PROGRAM Axis02_Status
VAR
//System_Bit
	Always_ON	:	BOOL	:=TRUE	;//상시 ON 
	Always_OFF	:	BOOL	:=FALSE	;//상시 OFF
	
//Motor_Command
	Axis02_Status_01: MC_ReadStatus;
	Axis02_Position_Read_01: MC_ReadActualPosition;
	Axis02_Velocity_Read_01: MC_ReadActualVelocity;
	Axis02_Reset_01: MC_Reset;
	Axis02_Stop_01: MC_Stop;
END_VAR

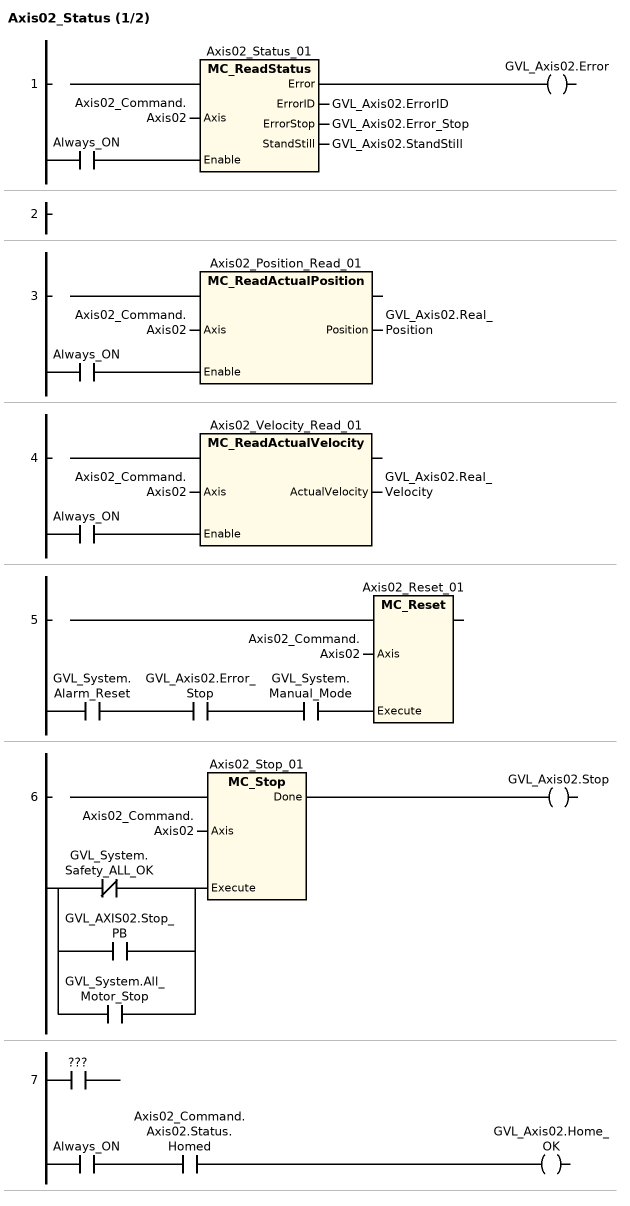
// NETWORK 1
Axis02_Status_01(
    Axis := Axis02_Command.Axis02,
    Enable := Always_ON,
    Error => GVL_Axis02.Error,
    ErrorID => GVL_Axis02.ErrorID,
    ErrorStop => GVL_Axis02.Error_Stop,
    StandStill => GVL_Axis02.StandStill); // MC_ReadStatus

// NETWORK 2

// NETWORK 3
Axis02_Position_Read_01(
    Axis := Axis02_Command.Axis02,
    Enable := Always_ON,
    Position => GVL_Axis02.Real_Position); // MC_ReadActualPosition

// NETWORK 4
Axis02_Velocity_Read_01(
    Axis := Axis02_Command.Axis02,
    Enable := Always_ON,
    ActualVelocity => GVL_Axis02.Real_Velocity); // MC_ReadActualVelocity

// NETWORK 5
Axis02_Reset_01(Axis := Axis02_Command.Axis02, Execute := GVL_System.Alarm_Reset AND GVL_Axis02.Error_Stop AND GVL_System.Manual_Mode); // MC_Reset

// NETWORK 6
Axis02_Stop_01(Axis := Axis02_Command.Axis02, Execute := NOT GVL_System.Safety_ALL_OK OR GVL_AXIS02.Stop_PB OR GVL_System.All_Motor_Stop); // MC_Stop
GVL_Axis02.Stop := Axis02_Stop_01.Done;

// NETWORK 7
GVL_Axis02.Home_OK := Always_ON AND Axis02_Command.Axis02.Status.Homed;

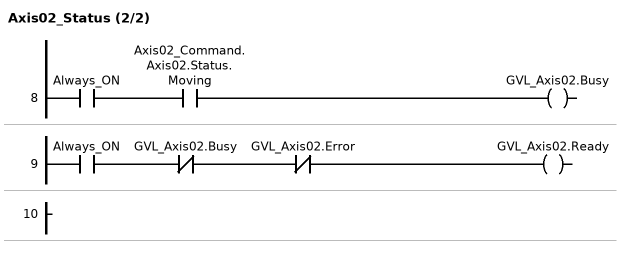
// NETWORK 8
GVL_Axis02.Busy := Always_ON AND Axis02_Command.Axis02.Status.Moving;

// NETWORK 9
GVL_Axis02.Ready := Always_ON AND NOT GVL_Axis02.Busy AND NOT GVL_Axis02.Error;

// NETWORK 10

END_PROGRAM

(* stored: Version 1.1.0.1, ProductVersion 3.1.4024.16
   POU Axis02_Status: Id {6c8f84cb-e148-4c91-9c9e-c81eb8526fa8}, SpecialFunc None *)
